FUNCTION_BLOCK PUBLIC FB_ALARM_INSTANCE
VAR_INPUT
	Alarm : REFERENCE TO FB_ALARM;
	Config : TYP_ALARM_CONFIG;
	State : E_ALARM_STATE;
END_VAR
VAR_OUTPUT
END_VAR
VAR
	_actDT : DT;
END_VAR

PROPERTY PUBLIC ActivationDateTime : DT
GET
ActivationDateTime := THIS^._actDT;
END_GET
SET
THIS^._actDT :=	ActivationDateTime;
END_SET
END_PROPERTY

METHOD PUBLIC Update : REFERENCE TO FB_ALARM_INSTANCE
VAR_INPUT
END_VAR
IF __ISVALIDREF(THIS^.Alarm) THEN
	THIS^.State := THIS^.Alarm.State;
END_IF;

Update REF= THIS^;
END_METHOD

PROPERTY PUBLIC VisuAlarm : TYP_VISU_ALARM
GET
VAR
	Alarm : TYP_VISU_ALARM;
END_VAR
Alarm.Code := THIS^.Config.Code;
Alarm.Priority := THIS^.Config.Priority;
Alarm.Message := THIS^.Config.Name;
Alarm.Name := THIS^.Config.Name;
Alarm.Timestamp := THIS^.ActivationDateTime;
Alarm.State := TO_STRING(THIS^.State);

VisuAlarm := Alarm;
END_GET
END_PROPERTY

END_FUNCTION_BLOCK

(* stored: Version 1.1.0.1, ProductVersion 3.1.4024.12
   POU FB_ALARM_INSTANCE: Id {f2324f30-a80f-4c23-8c09-e438e4b22386}, SpecialFunc None
   Property ActivationDateTime: Id {59cdcf77-47e1-48f5-96e0-6a47bf93abf8}
   Get Get: Id {435399f8-47a0-4a0a-bdb8-af5c45177d12}
   Set Set: Id {220516a4-cd6b-4537-bfa3-e9ee37d2bc6e}
   Method Update: Id {9219cb9e-ce21-40c6-b89a-2ef5b3bb50f3}
   Property VisuAlarm: Id {9e1e590a-a8a3-4469-9592-122ee15f4e75}
   Get Get: Id {aff9b831-cdf2-4600-99d3-40ede29cd463} *)
